// Brief: Master Arm Standby
FUNCTION_BLOCK PUBLIC FB_StateCtrlMountPanel EXTENDS FB_SlaveArmCtrlBase
VAR_INPUT
END_VAR
VAR_OUTPUT
END_VAR
VAR
END_VAR

METHOD PUBLIC init : BOOL
VAR_IN_OUT CONSTANT
	i_slaveArm	:FB_SlaveArm;
END_VAR
VAR_IN_OUT 
	r_slaveArmCtrlCmd :ST_SlaveArmCtrlCmds;
END_VAR
SUPER^.Init(i_slaveArm,r_slaveArmCtrlCmd);

// check if to hold the command joint position unchanged
checkToHoldLastCmds(i_slaveArm,r_slaveArmCtrlCmd);
END_METHOD

END_FUNCTION_BLOCK

(* stored: Version 1.1.0.1, ProductVersion 3.1.4024.12
   POU FB_StateCtrlMountPanel: Id {823d9da4-dfa7-45fa-b541-870812882ed0}, SpecialFunc None
   Method init: Id {ee3f7839-f2f4-4010-851e-5bc229c0ad27} *)
